{attribute 'qualified_only'}
VAR_GLOBAL
	Lh_full: BOOL;
	Lh_half: BOOL;
	Equal: BOOL;
	Rh_half: BOOL;
	Rh_full: BOOL;
	
	Lh_full_request: BOOL;
	Lh_half_request: BOOL;
	Equal_request: BOOL;
	Rh_half_request: BOOL;
	Rh_full_request: BOOL;
END_VAR

(* stored: Version 1.1.0.1, ProductVersion 3.1.4024.0
   GVL Torque_prediction: Id {a82d1187-fa61-4769-ac4a-437ad3831ad9} *)
